{attribute 'linkalways'} 
{attribute 'no_explicit_call' := 'This FB is a CLASS and must be accessed using methods or properties'}
{attribute 'enable_dynamic_creation'}
FUNCTION_BLOCK _BIT EXTENDS DatatypeBase implements I_BIT
VAR
	initialised : BOOL;
	activeParent : I_StructuredDatatype;
	activeByteOffset : PVOID;
	activeBitOffset : DWORD;
END_VAR

PROPERTY PUBLIC Address : PVOID
GET
IF NOT initialised THEN 
	RETURN;
END_IF

Address := activeParent.Address + activeByteOffset;
END_GET
END_PROPERTY

PROPERTY PUBLIC BitOffset : DWORD
GET
IF NOT initialised THEN 
	RETURN;
END_IF

BitOffset := activeBitOffset;
END_GET
END_PROPERTY

PROPERTY PUBLIC ByteOffset : PVOID
GET
IF NOT initialised THEN 
	RETURN;
END_IF

ByteOffset := activeByteOffset;
END_GET
END_PROPERTY

METHOD PUBLIC ClearReference
VAR_INPUT
END_VAR
activeParent := 0;
activeByteOffset := 0;
activeBitOffset := 0;
initialised := FALSE;
END_METHOD

METHOD PUBLIC Clone : I_Datatype
VAR
    pClone : POINTER TO _BIT;
END_VAR
pClone := __NEW(_BIT);

IF initialised THEN
	pClone^.MakeReferenceTo(activeParent, activeByteOffset, activeBitOffset);
END_IF

Clone := pClone^;
END_METHOD

METHOD PRIVATE GetBitValue : BOOL
VAR
	pByte : POINTER TO BYTE := Address;
END_VAR
IF NOT initialised THEN
	RETURN;
END_IF

CASE activeBitOffset OF
	0: GetBitValue := pByte^.0;
	1: GetBitValue := pByte^.1;
	2: GetBitValue := pByte^.2;
	3: GetBitValue := pByte^.3;
	4: GetBitValue := pByte^.4;
	5: GetBitValue := pByte^.5;
	6: GetBitValue := pByte^.6;
	7: GetBitValue := pByte^.7;
END_CASE;
END_METHOD

METHOD PUBLIC MakeReferenceTo
VAR_INPUT
	Parent : I_StructuredDatatype;
	ByteOffset : PVOID;
	BitOffset : DWORD;
END_VAR
activeParent := Parent;
activeByteOffset := ByteOffset;
activeBitOffset := BitOffset AND 16#7;
initialised := TRUE;
END_METHOD

PROPERTY PUBLIC Parent : I_StructuredDatatype
GET
Parent := activeParent;
END_GET
END_PROPERTY

METHOD PUBLIC SerializeWith
VAR_INPUT
	Serializer : I_Serializer;
END_VAR
Serializer.AddBool(GetBitValue());
END_METHOD

METHOD PRIVATE SetBitValue : BOOL
VAR_INPUT
	Value : BOOL;
END_VAR
VAR
	pByte : POINTER TO BYTE := Address;
END_VAR
IF NOT initialised THEN
	RETURN;
END_IF

CASE activeBitOffset OF
	0: pByte^.0 := Value;
	1: pByte^.1 := Value;
	2: pByte^.2 := Value;
	3: pByte^.3 := Value;
	4: pByte^.4 := Value;
	5: pByte^.5 := Value;
	6: pByte^.6 := Value;
	7: pByte^.7 := Value;
END_CASE;
END_METHOD

PROPERTY PUBLIC Size : UDINT
GET
Size := 1;
END_GET
END_PROPERTY

METHOD PUBLIC TryConvertTo : BOOL
VAR_INPUT
	Destination : ANY;
END_VAR
TryConvertTo := TryConvert_BOOL_To_Destination(Value, Destination);
END_METHOD

METHOD PUBLIC TryConvertTo_ : BOOL
VAR_INPUT
	Destination : I_Datatype;
END_VAR
VAR
	resultofBitConversion : BOOL;
	destinationAs_BIT : I_BIT;
	destinationAs_BOOL : I_BOOL;
	destinationAs_BYTE : I_BYTE;
	destinationAs_DINT : I_DINT;
	destinationAs_DT : I_DT;
	destinationAs_DWORD : I_DWORD;
	destinationAs_INT : I_INT;
	destinationAs_LINT : I_LINT;
	destinationAs_LREAL : I_LREAL;
	destinationAs_LWORD : I_LWORD;
	destinationAs_REAL : I_REAL;
	destinationAs_SINT : I_SINT;
	destinationAs_STRING : I_STRING;
	destinationAs_TOD : I_TOD;
	destinationAs_UDINT : I_UDINT;
	destinationAs_UINT : I_UINT;
	destinationAs_ULINT : I_ULINT;
	destinationAs_USINT : I_USINT;
	destinationAs_WORD : I_WORD;
END_VAR
IF destination.TryResolveAs_BIT(destinationAs_BIT) AND_THEN TryConvert_BOOL_TO_BOOL(Value, resultofBitConversion) THEN
	destinationAs_BIT.Value := resultOfBitConversion;
	TryConvertTo_ := TRUE;
	RETURN;
END_IF

IF destination.TryResolveAs_BOOL(destinationAs_BOOL) THEN
	TryConvertTo_ := TryConvert_BOOL_TO_BOOL(Value, destinationAs_BOOL.Value);
	RETURN;
END_IF
		
IF destination.TryResolveAs_BYTE(destinationAs_BYTE) THEN
	TryConvertTo_ := TryConvert_BOOL_TO_BYTE(Value, destinationAs_BYTE.Value);
	RETURN;
END_IF

IF destination.TryResolveAs_DINT(destinationAs_DINT) THEN
	TryConvertTo_ := TryConvert_BOOL_TO_DINT(Value, destinationAs_DINT.Value);
	RETURN;
END_IF

IF destination.TryResolveAs_DT(destinationAs_DT) THEN
	TryConvertTo_ := TryConvert_BOOL_TO_DT(Value, destinationAs_DT.Value);
	RETURN;
END_IF

IF destination.TryResolveAs_DWORD(destinationAs_DWORD) THEN
	TryConvertTo_ := TryConvert_BOOL_TO_DWORD(Value, destinationAs_DWORD.Value);
	RETURN;
END_IF

IF destination.TryResolveAs_INT(destinationAs_INT) THEN
	TryConvertTo_ := TryConvert_BOOL_TO_INT(Value, destinationAs_INT.Value);
	RETURN;
END_IF

IF destination.TryResolveAs_LINT(destinationAs_LINT) THEN
	TryConvertTo_ := TryConvert_BOOL_TO_LINT(Value, destinationAs_LINT.Value);
	RETURN;
END_IF

IF destination.TryResolveAs_LREAL(destinationAs_LREAL) THEN
	TryConvertTo_ := TryConvert_BOOL_TO_LREAL(Value, destinationAs_LREAL.Value);
	RETURN;
END_IF

IF destination.TryResolveAs_LWORD(destinationAs_LWORD) THEN
	TryConvertTo_ := TryConvert_BOOL_TO_LWORD(Value, destinationAs_LWORD.Value);
	RETURN;
END_IF

IF destination.TryResolveAs_REAL(destinationAs_REAL) THEN
	TryConvertTo_ := TryConvert_BOOL_TO_REAL(Value, destinationAs_REAL.Value);
	RETURN;
END_IF

IF destination.TryResolveAs_SINT(destinationAs_SINT) THEN
	TryConvertTo_ := TryConvert_BOOL_TO_SINT(Value, destinationAs_SINT.Value);
	RETURN;
END_IF

IF destination.TryResolveAs_STRING(destinationAs_STRING) THEN
	TryConvertTo_ := TryConvert_BOOL_TO_STRING(Value, destinationAs_STRING.Value);
	RETURN;
END_IF

IF destination.TryResolveAs_TOD(destinationAs_TOD) THEN
	TryConvertTo_ := TryConvert_BOOL_TO_TOD(Value, destinationAs_TOD.Value);
	RETURN;
END_IF

IF destination.TryResolveAs_UDINT(destinationAs_UDINT) THEN
	TryConvertTo_ := TryConvert_BOOL_TO_UDINT(Value, destinationAs_UDINT.Value);
	RETURN;
END_IF

IF destination.TryResolveAs_UINT(destinationAs_UINT) THEN
	TryConvertTo_ := TryConvert_BOOL_TO_UINT(Value, destinationAs_UINT.Value);
	RETURN;
END_IF

IF destination.TryResolveAs_ULINT(destinationAs_ULINT) THEN
	TryConvertTo_ := TryConvert_BOOL_TO_ULINT(Value, destinationAs_ULINT.Value);
	RETURN;
END_IF

IF destination.TryResolveAs_USINT(destinationAs_USINT) THEN
	TryConvertTo_ := TryConvert_BOOL_TO_USINT(Value, destinationAs_USINT.Value);
	RETURN;
END_IF

IF destination.TryResolveAs_WORD(destinationAs_WORD) THEN
	TryConvertTo_ := TryConvert_BOOL_TO_WORD(Value, destinationAs_WORD.Value);
	RETURN;
END_IF
END_METHOD

METHOD TryDeserializeFrom : BOOL
VAR_INPUT
	Deserializer : I_Deserializer;
	Feedback : I_DeserializerFeedback;
END_VAR
VAR 
	value : BOOL;
END_VAR
IF NOT Deserializer.TryGetBool(value, Feedback) THEN
	RETURN;
END_IF

SetBitValue(value);
TryDeserializeFrom := TRUE;
END_METHOD

METHOD TryMakeReferenceTo : BOOL
VAR_INPUT
	Target : I_Datatype;
END_VAR
VAR
	targetAsBit : I_BIT;
END_VAR
IF NOT Target.Root.TryResolveAs_BIT(targetAsBit) THEN
	RETURN;
END_IF

MakeReferenceTo(targetAsBit.Parent, targetAsBit.ByteOffset, targetAsBit.BitOffset);
TryMakeReferenceTo := TRUE;
END_METHOD

METHOD PUBLIC TryResolveAs_BIT : BOOL
VAR_INPUT
	Destination : REFERENCE TO I_BIT;
END_VAR
Destination := THIS^;
TryResolveAs_BIT := TRUE;
END_METHOD

PROPERTY PUBLIC TypeName : T_MAXSTRING
GET
TypeName := 'BIT';
END_GET
END_PROPERTY

PROPERTY PUBLIC Value : BOOL
GET
Value := GetBitValue();
END_GET
SET
SetBitValue(Value);
END_SET
END_PROPERTY

END_FUNCTION_BLOCK

(* stored: Version 1.1.0.1, ProductVersion 3.1.4024.15
   POU _BIT: Id {79c65b7e-7f7d-446e-a165-e9d39eed4032}, SpecialFunc None
   Folder Private: Id {6b544948-adc9-4ea0-aa46-ccb46a3a1863}
   Property Address: Id {24665800-2f18-474d-a292-e4b75def6510}
   Get Get: Id {fcd89903-c436-4c3b-ac93-f4ad730f61bf}
   Property BitOffset: Id {dbdaa237-0a72-420b-9700-970ae03a8397}
   Get Get: Id {a2a259b0-1c90-4795-9794-23537bb6d88d}
   Property ByteOffset: Id {7932e269-26c5-4045-b376-ab10e4abfb3c}
   Get Get: Id {7173f58b-74af-4a06-a8c2-960345c91948}
   Method ClearReference: Id {f4b37452-8608-46e6-b355-3636a938af92}
   Method Clone: Id {ddb8f313-987b-4d70-b0d6-6ef005159f0e}
   Method GetBitValue: Id {4f9ceb2e-0758-4d8c-b49e-2fcdbcaaad48}
   Method MakeReferenceTo: Id {aa5cee22-3980-4a33-9855-8cf108d9f1d5}
   Property Parent: Id {e7f6c8e9-8881-4d9c-b9a2-3f79f5916f52}
   Get Get: Id {8f809583-6878-468e-8d7c-b90be9df712d}
   Method SerializeWith: Id {124e1cba-b0c7-4c18-9448-c4229ffb9e59}
   Method SetBitValue: Id {43f501b1-a1c7-4e08-9bf7-144d284db803}
   Property Size: Id {858d638c-8af0-47ed-90fa-b9d90b10dace}
   Get Get: Id {c7e65aff-e45c-41be-9deb-8ac8d0044487}
   Method TryConvertTo: Id {c73b74c6-8171-0676-2782-c0e364cf4731}
   Method TryConvertTo_: Id {0aab26e9-f98c-02cf-0fcb-3427c84069f9}
   Method TryDeserializeFrom: Id {d7a623ef-3a27-44f3-98f8-9fe9f95aaeec}
   Method TryMakeReferenceTo: Id {20df3f08-9c63-4138-86d5-f858191770d5}
   Method TryResolveAs_BIT: Id {42135720-d2a0-080c-2613-4773f8581ae0}
   Property TypeName: Id {a96405b3-76e7-4582-9617-d689a46afdea}
   Get Get: Id {9fa59ead-7968-4b99-b49a-fe8ba877b032}
   Property Value: Id {4414726e-2e53-4422-ad51-ffff582d7103}
   Get Get: Id {b818634b-a990-4956-aec7-81f0002a3caa}
   Set Set: Id {52e4f29f-75b2-4dba-98b5-6e9057353529} *)
